        IF NOT _done THEN
            _sut_A.SequenceRun := _plcCycleCounter;
            _sut_N.SequenceRun := _plcCycleCounter;
            _sut_A._RunExecutionSubstitute();
            _sut_N._RunExecutionSubstitute();
            _sut_A.SaveNumberOfStepsInSequence();
            _sut_N.SaveNumberOfStepsInSequence();
        END_IF

        _done := _plcCycleCounter >= 2 * _cyclicCycles + _stepInEvents + 1;
        ProbeDoneWhen(_done);
{endregion}
	 eTcoSequenceTests.MissedSequenceOpening:
	    _sut_A.Restore();
	 	THIS^._Open();
	 	_sut_A.Step(10, TRUE, '');
		THIS^._Close();
		THIS^.ProbeDoneWhen(TRUE);
	 eTcoSequenceTests.MissedSequenceClosing:
	 	_sut_A.Restore();
	 	THIS^._Open();
	    _sut_A.Open();
	 	_sut_A.Step(10, TRUE, '');
		THIS^._Close();
		_sut_A.Messenger.Clear();
		THIS^._Open();
		 _sut_A.Open();
		_sut_A.Step(10, TRUE, '');
		THIS^.ProbeDoneWhen(TRUE);
	eTcoSequenceTests.FreshStateEntry:
		
		THIS^._sut_A.Open();
		IF(_sut_A.Step(10, TRUE, 'ENTER AND LEAVE')) THEN
			THIS^.FreshStateEntry_enter_and_leave_must_be_true := _sut_A.IsFreshState;
			_sut_A.CompleteStep(); 			 
		END_IF;
		
		IF(_sut_A.Step(20, TRUE, 'ENTER MULTIPLE CYCLES')) THEN 
			IF(FreshStateEntry_counter = 0) THEN
				THIS^.FreshStateEntry_enter_and_two_cycles_on_first_must_be_true := _sut_A.IsFreshState;
			END_IF;				
			THIS^.FreshStateEntry_enter_and_two_cycles_on_second_must_be_false := _sut_A.IsFreshState;
			_sut_A.StepCompleteWhen(FreshStateEntry_counter = 1);
			FreshStateEntry_counter := FreshStateEntry_counter + 1;
		END_IF;
		
		IF(_sut_A.Step(40, TRUE, 'ENTER MULTIPLE CYCLES')) THEN 						
			FreshStateEntry_on_multiple_calls_but_not_first_must_be_false := _sut_A.IsFreshState;											
			FreshStateEntry_counter := FreshStateEntry_counter + 1;
			_sut_A.StepCompleteWhen(FreshStateEntry_counter = 100);
		END_IF;
		
		IF(_sut_A.Step(50, TRUE, 'ENTER MULTIPLE CYCLES')) THEN
			FreshStateEntry_on_request_step_single_call_must_be_true :=	_sut_A.IsFreshState;		 			
			_sut_A.CompleteStep();
			IF(FreshStateEntry_counter = 0) THEN
				_sut_A.RequestStep(70);
			END_IF
		END_IF;
		
		IF(_sut_A.Step(60, TRUE, 'ENTER MULTIPLE CYCLES')) THEN					 			
			_sut_A.RequestStep(50);
			FreshStateEntry_counter := 0;
		END_IF;
		
		IF(_sut_A.Step(70, TRUE, 'ENTER MULTIPLE CYCLES')) THEN					 			
			THIS^.ProbeDoneWhen(TRUE);
		END_IF;
		
		THIS^._sut_A.Close();
END_CASE
END_METHOD

METHOD INTERNAL ReadOutCycleCounters
_startCycles		:=		THIS^.StartCycleCount;
_endCycles			:=		THIS^.EndCycleCount;

_myIdentity			:= 		THIS^.Identity;
END_METHOD

END_FUNCTION_BLOCK

(* stored: Version 1.1.0.1
   POU TcoSequenceTestContext: Id {356b8118-7b52-0b5a-1d80-284c7dd3d13f}, SpecialFunc None
   Method _ClearPlcCycleCounter: Id {24e04400-21af-0e40-1dc6-243e032ffa21}
   Method Main: Id {06e1f7c7-c7b2-044c-3ea8-d39a941ddbe3}
   Method ReadOutCycleCounters: Id {d4aea31d-39d8-0427-14ad-84c644f2dd25} *)
